FUNCTION_BLOCK FB_MovAvg
VAR_INPUT
	i_rIn : LREAL;
	i_nSamples : UINT;
END_VAR
VAR_OUTPUT
	o_rOut : LREAL;
END_VAR
VAR
	s_nSampleCounter : UINT;
END_VAR

END_FUNCTION_BLOCK

(* stored: Version 1.1.0.1, ProductVersion 3.1.4024.12
   POU FB_MovAvg: Id {94161948-1aa6-4a27-a829-3f9dbd183760}, SpecialFunc None *)
